PROGRAM MAIN
VAR
	StepAxis	:	AXIS_REF;
	ServoAxis	:	AXIS_REF;
	fbCoupling	:	FB_Coupling;
	fbMqtt		:	FB_MQTT;
	fbSequence	:	FB_Sequence;
END_VAR


fbMqtt();
GVL_PLC.lrActPosition := ServoAxis.NcToPlc.ActPos;

fbSequence(ServoAxis:=ServoAxis,StepAxis:=StepAxis);

ServoAxis();
StepAxis();

END_PROGRAM

(* stored: Version 1.1.0.1, ProductVersion 3.1.4024.13
   POU MAIN: Id {f5bd4718-2552-47f9-921d-cb1f6b642716}, SpecialFunc None *)
